FUNCTION_BLOCK "CylindersMain"
{ S7_Optimized_Access := 'TRUE' }
VERSION : 0.1
   VAR
      res : Bool;
   END_VAR


BEGIN

	"CylinderGeneratedCalls_DB"();

	"CylinderCollisions"();

	"CylindersHMIMessage"(CylinderNumber=>"CylindersHMI".CylinderInfoHMI,
	                      CylinderAction=>"CylindersHMI".CylinderInfoHMIAction);

END_FUNCTION_BLOCK

